// TIA Portal V20 export
DATA_BLOCK "Appo"   // DB2
TITLE = Variabili di appoggio
{ S7_Optimized_Access := 'TRUE' }
// Per spostare dati nel sw in modo facile
// stored: MemoryReserve 100
   VAR
      Gt1St : Byte;
   END_VAR
BEGIN
END_DATA_BLOCK
